// TIA Portal V20 export
TYPE "typeEm4MonitoringCmStatus"
// stored: Access Published, Namespace Unit1
   STRUCT
      compAxis { ExternalWritable := 'False'} : "LBC_typeAxisControlNodeMonitoring";
      feedRollAxis { ExternalWritable := 'False'} : "LBC_typeAxisControlNodeMonitoring";
      cutterAxis { ExternalWritable := 'False'} : "LBC_typeAxisControlNodeMonitoring";
      moveAxis { ExternalWritable := 'False'} : "LBC_typeAxis64PosControlNodeMonitoring";
      feederCyl { ExternalWritable := 'False'} : "LBC_typeTwoWayActuatorControlNodeMonitoring";
      compSafetyPin { ExternalWritable := 'False'} : "LBC_typeDigitalSignalControlNodeMonitoring";
   END_STRUCT;
END_TYPE
